FUNCTION_BLOCK FB_TcpBlock
VAR
	tcpTime : TIMESTRUCT;
	
	dataType : (NO_DATA, BUNDLE_TRANSFER, BUNDLE_ETA, GENERAL_EVENT);
	timestamp : TIMESTRUCT;
	
	binaryData : ARRAY[0..50000] OF BYTE;
	jsonData : STRING(2000);
	xmlData : STRING(2000);
END_VAR

METHOD sendBundleETA : BOOL
VAR_INPUT
	eta : TIMESTRUCT;
	bundleId : STRING;
END_VAR
END_METHOD

METHOD sendBundleTransfer : BOOL
VAR_INPUT
END_VAR
END_METHOD

METHOD setTcpTime : BOOL
tcpTime := GVL.systemTime;
END_METHOD

END_FUNCTION_BLOCK

(* stored: Version 1.1.0.1, ProductVersion 3.1.4024.11
   POU FB_TcpBlock: Id {93959326-5c29-4289-af5b-7e33722a43ea}, SpecialFunc None
   Method sendBundleETA: Id {ffb937b3-abc3-4f36-acf7-0a4a4f58dada}
   Method sendBundleTransfer: Id {4de91b01-6aeb-44f5-8304-79e331fb683a}
   Method setTcpTime: Id {94cb8c6e-87a2-4e85-90be-8604d19d3807} *)
